TYPE T_Ctrl_SIf_STB_Cur :
STRUCT
	/// Hangers passed total counter (reset in state OFF)
	dinHangersPassedTotal: DINT;
	/// Hangers passed package counter (is updated when “RELEASE_ALL” command is completed)
	dinHangersPassedPackage: DINT;
	/// Hanger detected
	bolHangerDetected: BOOL;
	/// Approximate number of hangers in buffer
	dinNumOfHangersInBuffer: DINT;
	/// Buffer is full
	bolBufferFull: BOOL;
END_STRUCT
END_TYPE

(* stored: Version 1.1.0.1, ProductVersion 3.1.0.19
   DUT T_Ctrl_SIf_STB_Cur: Id {31d9788b-af4e-4154-b282-f4a1ef5d912d} *)
